// TIA Portal V17 export
// export: Created 2023-02-14T02:49:28.8134526Z, ExportSetting WithDefaults, DisplayName Totally Integrated Automation Portal, DisplayVersion V17, DisplayName TIA Portal Openness, DisplayVersion V17, DisplayName TIA Portal Teamcenter Gateway, DisplayVersion V17, DisplayName TIA Portal Version Control Interface, DisplayVersion V17, DisplayName SINAMICS Startdrive Advanced, DisplayVersion V17, DisplayName SINAMICS Startdrive G130, G150, S120, S150, SINAMICS MV, S210, DisplayVersion V17, DisplayName SINAMICS Startdrive G110M, G120, G120C, G120D, G120P, G115D, DisplayVersion V17, DisplayName STEP 7 Professional, DisplayVersion V17, DisplayName STEP 7 Safety, DisplayVersion V17, DisplayName WinCC Professional, DisplayVersion V17
DATA_BLOCK "IO_Valve_Blend21_DB"   // DB39
VERSION : 0.1
// stored: AutoNumber true, DBAccessibleFromOPCUA true, DBAccessibleFromWebserver true, InstanceOfName IO_Valve_Blend21, InstanceOfType FB
"IO_Valve_Blend21"
   // VAR_INPUT
   //    "lock 1" : Bool;
   //    "lock 2" : Bool;
   //    "lock 3" : Bool;
   //    "lock 4" : Bool;
   //    init : Bool;
   //    reset : Bool;
   //    testing : Bool;
   // END_VAR
   // VAR
   //    "AV-21.01" : "Valve";
   //    "AV-21.02" : "Valve";
   //    "AV-21.03" : "Valve";
   //    "AV-21.04" : "Valve";
   //    "AV-21.05" : "Valve";
   //    "AV-21.06" : "Valve";
   //    "AV-21.07" : "Valve";
   //    "AV-21.08" : "Valve";
   //    "AV-21.09" : "Valve";
   //    "AV-21.10" : "Valve";
   //    "AV-21.11" : "Valve";
   //    "AV-21.21" : "Valve";
   //    "AV-21.22" : "Valve";
   //    "AV-21.23" : "Valve";
   //    "AV-21.24" : "Valve";
   //    "AV-21.25" : "Valve";
   //    "AV-21.26" : "Valve";
   //    "AV-21.27" : "Valve";
   //    "AV-21.28" : "Valve";
   //    "AV-21.29" : "Valve";
   //    "AV-21.30" : "Valve";
   //    "AV-21.31" : "Valve";
   //    "AV-21.32" : "Valve";
   //    "AV-21.33" : "Valve";
   //    "AV-21.34" : "Valve";
   //    "AV-21.35" : "Valve";
   //    "AV-21.41" : "Valve";
   //    "AV-21.42" : "Valve";
   // END_VAR
BEGIN
END_DATA_BLOCK
